// TIA Portal V19 export
FUNCTION "PosAxisToPosMat_Wheel" : LReal   // FC104, LAD
TITLE = From pos axis to pos material
// stored: Access Published, SetENOAutomatically false
   VAR_INPUT
      PosAxis : LReal;
      Data : "MatCountData";
   END_VAR
   VAR_TEMP
      HalfModule : LReal;
      HalfNegativeModule : LReal;
      DeltaPosAx : LReal;
      DeltaMatCounter : LReal;
      MatCountPosCandidate : LReal;
   END_VAR
BEGIN

REGION Network 1: Half MODULE
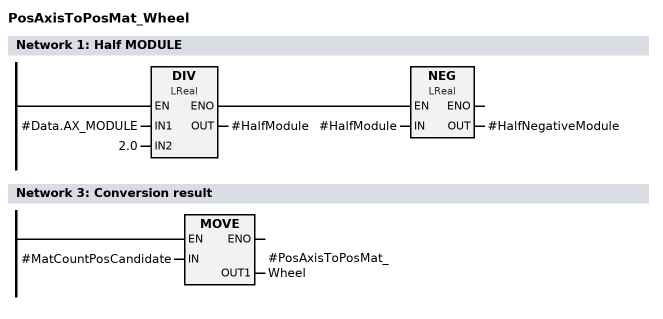
   RUNG wire#powerrail
      { S7_Templates := "SrcType := LReal" } Div(in1 := #Data.AX_MODULE, in2 := 2.0, out => #HalfModule)
      { S7_Templates := "SrcType := LReal" } Neg(in := #HalfModule, out => #HalfNegativeModule)
   END_RUNG
   // the same network as SCL:
   #HalfModule := #Data.AX_MODULE / 2.0;
   #HalfNegativeModule := -#HalfModule;
END_REGION

REGION Network 2 (SCL): Calculate position
   #DeltaPosAx := #PosAxis - #Data.AxPositionPrevious;

   IF #DeltaPosAx > #HalfModule THEN
       #DeltaPosAx := #DeltaPosAx - #Data.AX_MODULE;
   ELSIF #DeltaPosAx < #HalfNegativeModule THEN
       #DeltaPosAx := #DeltaPosAx + #Data.AX_MODULE;
   END_IF;

   #DeltaMatCounter := #DeltaPosAx * #Data.FAK;
   #MatCountPosCandidate := #Data.CounterValue + #DeltaMatCounter;

   IF #MatCountPosCandidate >= #Data.COUNTER_MODULE THEN
       #MatCountPosCandidate := #MatCountPosCandidate - #Data.COUNTER_MODULE;
   ELSIF #MatCountPosCandidate < 0.0 THEN
       #MatCountPosCandidate := #MatCountPosCandidate + #Data.COUNTER_MODULE;
   END_IF;

   IF ABS_LREAL(#MatCountPosCandidate - #Data.COUNTER_MODULE) < 0.01 THEN
       #MatCountPosCandidate := 0.0;
   END_IF;
END_REGION

REGION Network 3: Conversion result
   RUNG wire#powerrail
      Move(in := #MatCountPosCandidate, out1 => #PosAxisToPosMat_Wheel)
   END_RUNG
   // the same network as SCL:
   #PosAxisToPosMat_Wheel := #MatCountPosCandidate;
END_REGION
END_FUNCTION
